// TwinCAT 3 PLC project VISU
// ProgramVersion: 3.1.4022.2
// libraries:
//   Tc2_Database, * (Beckhoff Automation GmbH)
//   Tc2_Standard, * (Beckhoff Automation GmbH)
//   Tc2_System, * (Beckhoff Automation GmbH)
//   Tc3_Database, * (Beckhoff Automation GmbH)
//   Tc3_EventLogger, * (Beckhoff Automation GmbH)
//   Tc3_IotBase, * (Beckhoff Automation GmbH)
//   Tc3_Module, * (Beckhoff Automation GmbH)
// project tree:
//   DUTs/ ST_Record.TcDUT
//   / GlobalTextList.TcGTLO, PlcTask.TcTTO, Visualization Manager.TcVMO (not stored), VISU_TASK.TcTTO
//   GVLs/ GVL.TcGVL
//   POUs/ MAIN.TcPOU, PROG_ReadStructure.TcPOU
//   VISUs/ Visualization.TcVIS

CONFIGURATION VISU
    RESOURCE PLC ON TwinCAT3
        TASK PlcTask(INTERVAL := T#10ms, PRIORITY := 20);
        TASK VISU_TASK(INTERVAL := T#200000us, PRIORITY := 30);
        PROGRAM MAIN WITH PlcTask : MAIN;
        PROGRAM VisuElems_Visu_Prg WITH VISU_TASK : VisuElems.Visu_Prg;
    END_RESOURCE
END_CONFIGURATION

// ---- DUTs/ST_Record.TcDUT
TYPE ST_Record :
STRUCT
	nID : LINT;
	tTimestamp : DATE_AND_TIME;
	rSinValue : REAL;
END_STRUCT
END_TYPE

// ---- GVLs/GVL.TcGVL
{attribute 'qualified_only'}
VAR_GLOBAL
	rSinValue : REAL;
	aReadStruct : ARRAY[0..200] OF ST_Record;
	
END_VAR

// ---- POUs/MAIN.TcPOU
PROGRAM MAIN
VAR
	v : INT := 0;
END_VAR

v := v+1;
PROG_ReadStructure();

END_PROGRAM

// ---- POUs/PROG_ReadStructure.TcPOU
PROGRAM PROG_ReadStructure
VAR
	fbSqlResult : FB_SQLResult(sNetID := '', tTimeout := T#5S);
	nState : INT := 0;

	aReadStruct2 : ARRAY[0..9] OF ST_Record;
	aReadStruct3 : ST_Record;
	aReadStruct4 : ST_Record;
	aReadStruct5 : ST_Record;
	
	fbPLCDBRead : FB_PLCDBRead (sNetID := '', tTimeout := T#5S);
	
	fbPLCDBWrite    :  FB_PLCDBWrite(sNetID := '', tTimeout := T#5S);
	ColumnNames : ARRAY[0..3] OF STRING(50);
	res : Tc3_EventLogger.I_TcResultEvent;
	res2 : UDINT;
	res3 : WSTRING(255);
	res4 : T_MaxString;
	res5 : WSTRING(255);
	res6 : E_Severity;
	
	
	bSetParameter : BOOL := TRUE;
	nCount: INT;
	
	fbPLCDBCmd       : FB_PLCDBCmd(sNetID := '', tTimeout := T#5S);
	
	 sCmd             : STRING (1000); 
	 nRecords         : UDINT := 1;
	// myStruct         : ST_DataAll;
	fbTimer : TON := (PT:=T#2S);
	
	startIndex: INT := 4;
	
	sCzas : STRING;
END_VAR



IF bSetParameter THEN
	bSetParameter := FALSE;
	// get values from internal tc db srv storage 
	ColumnNames[0] := 'ID';
	ColumnNames[1] := 'Timestamp';
	ColumnNames[2] := 'Message';
	aReadStruct4.nID := 11;
	aReadStruct4.rSinValue := 666;
	aReadStruct4.tTimestamp := DT#1970-01-01-00:00;
	
	nState := 20;
	nCount := 0;
END_IF


fbTimer(IN:=TRUE);
IF fbTimer.Q THEN // publish new payload every second
	fbTimer(IN:=FALSE);
	startIndex := startIndex+1;
	nState := 20;
	
END_IF


// set command with placeholder
sCmd := 'SELECT ID,	Timestamp,	Message FROM 	table4_autoIncrement';
//nState := 20;
// call functionblock

IF nState = 20 THEN
	IF fbPLCDBCmd.ExecuteDataReturn(
		hDBID:= 1, 
		pExpression:= ADR(sCmd), 
		cbExpression:= SIZEOF(sCmd), 
		pData:= 0, 
		cbData:= 0, 
		pParameter:= 0, 
		cbParameter:= 0,
		nStartIndex:= nRecords-1 , 
		nRecordCount:= 10, 
		pReturnData:= ADR(aReadStruct5), 
		cbReturnData:= SIZEOF(aReadStruct5), 
		pRecords:= ADR(nRecords)) 
	THEN
		IF fbPLCDBCmd.bError THEN
			nState := 255; 
		ELSE
			aReadStruct3 := aReadStruct5;
			sCzas := DT_TO_STRING(aReadStruct3.tTimestamp);
			nState := 10;
		END_IF
	END_IF
END_IF

END_PROGRAM

// ---- GlobalTextList.TcGTLO
TEXTLIST GlobalTextList
  233 = '%'
  883 = '%2.5f'
  242 = '%f'
  247 = '%s'
  410 = "%t['Last update:' ddd MMM dd.MM.yy 'at' HH:mm:ss]"
  688 = "%t['Last update:'dd.MM.yy 'at' HH:mm:ss]"
  923 = 'Czas: %s'
  29 = 'd'
  16 = 'f'
  295 = 'ID: %d'
  193 = 'LABEL'
  483 = 'PROG_ReadStructure.aReadStruct2.tTimestamp'
END_TEXTLIST

// ---- VISUs/Visualization.TcVIS
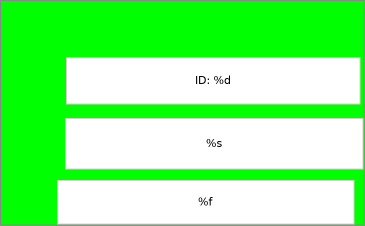
VISUALIZATION Visualization  // 365x226
    Textfield (57,180 297x44), "%f", text variable: PROG_ReadStructure.aReadStruct3.rSinValue
    Textfield (65,118 298x51), "%s", text variable: PROG_ReadStructure.sCzas
    Textfield (66,57 294x47), "ID: %d", text variable: PROG_ReadStructure.aReadStruct3.nID
END_VISUALIZATION
